// TIA Portal V15.1 export
// export: Created 2024-05-17T05:38:46.400505Z, ExportSetting WithDefaults, DisplayName Totally Integrated Automation Portal, DisplayVersion V15.1 Update 5, DisplayName TIA Portal Openness, DisplayVersion V15.1 Update 5, DisplayName SINAMICS Startdrive Advanced, DisplayVersion V15.1, DisplayName G130, G150, S120, S150, SINAMICS MV, S210, DisplayVersion V15.1, DisplayName G110M, G120, G120C, G120D, G120P, DisplayVersion V15.1, DisplayName STEP 7 Professional, DisplayVersion V15.1 Update 5, DisplayName STEP 7 Safety, DisplayVersion V15.1, DisplayName WinCC Professional, DisplayVersion V15.1 Update 5, DisplayName SIMATIC Visualization Architect, DisplayVersion V15.1
FUNCTION_BLOCK "LGBRollerDoorIO"   // FB6674, FBD
TITLE = LGBRollerDoorIO
{ S7_Optimized_Access := 'TRUE' }
VERSION : 0.1
// stored: AutoNumber false, IsIECCheckEnabled false, IsRetainMemResEnabled false, MemoryReserve 100, SetENOAutomatically False, UDAEnableTagReadback false
   VAR_INPUT
      I_DoorOpened { ExternalAccessible := 'False'; ExternalVisible := 'False'; ExternalWritable := 'False'} : Bool;   // Position Set detection or summary / Door Opened
      I_DoorClosed { ExternalAccessible := 'False'; ExternalVisible := 'False'; ExternalWritable := 'False'} : Bool;   // Position Reset detection or summary / Door Closed
      I_DoorClosedSafety { ExternalAccessible := 'False'; ExternalVisible := 'False'; ExternalWritable := 'False'} : Bool;   // Position Reset detection or summary / Door Closed Safety signal
      I_Ready { ExternalAccessible := 'False'; ExternalVisible := 'False'; ExternalWritable := 'False'} : Bool;   // Device Ready
      I_EnableAlarm { ExternalAccessible := 'False'; ExternalVisible := 'False'; ExternalWritable := 'False'} : Bool;   // Enable alarm / Enable Alarm
      I_MotorProtection { ExternalAccessible := 'False'; ExternalVisible := 'False'; ExternalWritable := 'False'} : Bool;   // Motor protection
      I_OpenBegin { ExternalAccessible := 'False'; ExternalVisible := 'False'; ExternalWritable := 'False'} : Bool;   // Function Set begin selection / Function Open begin selection
      I_CloseBegin { ExternalAccessible := 'False'; ExternalVisible := 'False'; ExternalWritable := 'False'} : Bool;   // Function Reset begin selection / Function Close begin selection
      I_CmdOpenIntlkOK { ExternalAccessible := 'False'; ExternalVisible := 'False'; ExternalWritable := 'False'} : Bool;   // Set Interlock / Command Open Interlock
      I_CmdCloseIntlkOK { ExternalAccessible := 'False'; ExternalVisible := 'False'; ExternalWritable := 'False'} : Bool;   // Reset Interlock / Command Close Interlock
      I_PBSet { ExternalAccessible := 'False'; ExternalVisible := 'False'; ExternalWritable := 'False'} : Bool;   // Push button for Set direction (used in manual with button OP panels )
      I_PBReset { ExternalAccessible := 'False'; ExternalVisible := 'False'; ExternalWritable := 'False'} : Bool;   // Push button for reset direcion (used in manual with pushbutton OP panels) / Push button for Reset direction (used in manual with Pushbutton OP panels)
      I_SafetyOk { ExternalAccessible := 'False'; ExternalVisible := 'False'; ExternalWritable := 'False'} : Bool;   // Safety Ok
      C_MotorProtectionNc { ExternalAccessible := 'False'; ExternalVisible := 'False'; ExternalWritable := 'False'} : Bool;   // Motor Protection Normally closed
      C_EnalbeRepatAlarmBypass { ExternalAccessible := 'False'; ExternalVisible := 'False'; ExternalWritable := 'False'} : Bool;   // Enable repeat alarm Bypass active
      C_RepeatAlarmBypass { ExternalAccessible := 'False'; ExternalVisible := 'False'; ExternalWritable := 'False'} : Time;   // Time to repeat alarm Bypass is active
   END_VAR
   VAR_OUTPUT
      O_CmdOpen { ExternalAccessible := 'False'; ExternalVisible := 'False'; ExternalWritable := 'False'} : Bool;   // Command to activate Set movement / Command to Activate Set movement / Command to Activate Open movement
      O_CmdClose { ExternalAccessible := 'False'; ExternalVisible := 'False'; ExternalWritable := 'False'} : Bool;   // Command to activate Reset movement / Command to Activate Reset movement / Command to Activate Close movement
      O_DoorOpened { ExternalAccessible := 'False'; ExternalVisible := 'False'; ExternalWritable := 'False'} : Bool;   // Door Opened
      O_DoorClosed { ExternalAccessible := 'False'; ExternalVisible := 'False'; ExternalWritable := 'False'} : Bool;   // Door Closed
      O_FuncRunning { ExternalAccessible := 'False'; ExternalVisible := 'False'; ExternalWritable := 'False'} : Bool;   // Signal that the function is busy
      O_LEDOpen { ExternalAccessible := 'False'; ExternalVisible := 'False'; ExternalWritable := 'False'} : Bool;   // Ledindication / Led indication for Open
      O_LEDClose { ExternalAccessible := 'False'; ExternalVisible := 'False'; ExternalWritable := 'False'} : Bool;   // Ledindication / Led indication for Close
      O_AlarmABCondition { ExternalAccessible := 'False'; ExternalVisible := 'False'; ExternalWritable := 'False'} : Bool;   // Alarms AB condition
      O_AlarmA { ExternalAccessible := 'False'; ExternalVisible := 'False'; ExternalWritable := 'False'} : Bool;   // Summation Alarm A of roller. / Alarm A
      O_AlarmB { ExternalAccessible := 'False'; ExternalVisible := 'False'; ExternalWritable := 'False'} : Bool;   // Summation Alarm B of roller. / Alarm B
      O_AlarmC { ExternalAccessible := 'False'; ExternalVisible := 'False'; ExternalWritable := 'False'} : Bool;   // Summation Alarm C of roller. / Alarm C
      O_AlarmD { ExternalAccessible := 'False'; ExternalVisible := 'False'; ExternalWritable := 'False'} : Bool;   // Summation Alarm D of roller. / Alarm D
      H_AlarmDWord { ExternalAccessible := 'False'; ExternalVisible := 'False'; ExternalWritable := 'False'} : DWord;   // HMI Animation of the alarms of the roller / HMI Animation
   END_VAR
   VAR_IN_OUT
      IO_GroupInterlock { ExternalAccessible := 'False'; ExternalVisible := 'False'; ExternalWritable := 'False'} : Bool;   // Is this OP selected? Refers to the interlocking word of this group
      IO_Modes : "Modes";
      H_HMI : "H_HMI";   // Animation
      H_RollerDoorIO : "H_GBRollerDoorIO";   // Animation
   END_VAR
   VAR
      AA_MotorProtectionAlm { ExternalAccessible := 'False'; ExternalVisible := 'False'; ExternalWritable := 'False'} : Bool;   // Motor protection alarm / Motor protection Alarm
      AB_DoorClosedSafety { ExternalAccessible := 'False'; ExternalVisible := 'False'; ExternalWritable := 'False'} : Bool;   // Safety Switch alarm / Safety Switch Alarm / Door is closed but the safety signal 'Door Closed' is missing
      AB_DoorClosedNotSafety { ExternalAccessible := 'False'; ExternalVisible := 'False'; ExternalWritable := 'False'} : Bool;   // Safety Switch alarm / Safety Switch Alarm / Door is closed but the NOT safety signal 'Door Closed' is missing
      AC_NotReadyAlm { ExternalAccessible := 'False'; ExternalVisible := 'False'; ExternalWritable := 'False'} : Bool;   // Not Ready To Run / Ej Drift Klar
      AC_OutOfUse { ExternalAccessible := 'False'; ExternalVisible := 'False'; ExternalWritable := 'False'} : Bool;   // The bypass is active, door is Out of Use (stay ALL the time open)
      AD_IntlkOpenAlm { ExternalAccessible := 'False'; ExternalVisible := 'False'; ExternalWritable := 'False'} : Bool;   // Alarm interlock Set / Alarm Interlock Set / Alarm Interlock Command Open
      AD_IntlkCloseAlm { ExternalAccessible := 'False'; ExternalVisible := 'False'; ExternalWritable := 'False'} : Bool;   // Alarm interlock Reset / Alarm Interlock Reset / Alarm Interlock Command Close
      AlarmA { ExternalAccessible := 'False'; ExternalVisible := 'False'; ExternalWritable := 'False'} : Bool;   // Summation Alarm A
      AlarmB { ExternalAccessible := 'False'; ExternalVisible := 'False'; ExternalWritable := 'False'} : Bool;   // Summation Alarm B
      AlarmC { ExternalAccessible := 'False'; ExternalVisible := 'False'; ExternalWritable := 'False'} : Bool;   // Summation Alarm C
      AlarmD { ExternalAccessible := 'False'; ExternalVisible := 'False'; ExternalWritable := 'False'} : Bool;   // Summation Alarm D
      FuncRunning { ExternalAccessible := 'False'; ExternalVisible := 'False'; ExternalWritable := 'False'} : Bool;   // Function running
      AlarmCondMotorProtection { ExternalAccessible := 'False'; ExternalVisible := 'False'; ExternalWritable := 'False'} : Bool;   // Alarm condition
      AlarmCondDoorClosedSafety { ExternalAccessible := 'False'; ExternalVisible := 'False'; ExternalWritable := 'False'} : Bool;   // Alarm condition
      AlarmCondDoorClosedNotSafety { ExternalAccessible := 'False'; ExternalVisible := 'False'; ExternalWritable := 'False'} : Bool;   // Alarm condition
      IntlkOpenAlmCond { ExternalAccessible := 'False'; ExternalVisible := 'False'; ExternalWritable := 'False'} : Bool;   // Alarm interlock Set condition / Alarm Interlock Set condition / Alarm Interlock Open condition
      IntlkCloseAlmCond { ExternalAccessible := 'False'; ExternalVisible := 'False'; ExternalWritable := 'False'} : Bool;   // Alarm interlock Reset condition / Alarm Interlock Reset condition / Alarm Interlock Close condition
      CmdOpen { ExternalAccessible := 'False'; ExternalVisible := 'False'; ExternalWritable := 'False'} : Bool;   // Command set / Command Open Door
      CmdClose { ExternalAccessible := 'False'; ExternalVisible := 'False'; ExternalWritable := 'False'} : Bool;   // Dommand reset / DCommand Reset / Command Close Door
      AlarmABCondition { ExternalAccessible := 'False'; ExternalVisible := 'False'; ExternalWritable := 'False'} : Bool;   // Alarm AB condition / Alarm AB Condition
   END_VAR
   VAR DB_SPECIFIC
      OpenCloseOutOfUse { ExternalAccessible := 'False'; ExternalVisible := 'False'; ExternalWritable := 'False'} : Bool;   // Status door by Out of Use
      Edge { ExternalAccessible := 'False'; ExternalVisible := 'False'; ExternalWritable := 'False'} : Array[0..10] of Bool;   // Edge
   END_VAR
   VAR
      T_DoorClosedSafety { ExternalAccessible := 'False'; ExternalVisible := 'False'; ExternalWritable := 'False'} : IEC_TIMER;   // On Delay Timer Safety signal
      T_DoorClosedNotSafety { ExternalAccessible := 'False'; ExternalVisible := 'False'; ExternalWritable := 'False'} : IEC_TIMER;   // On Delay Timer Safety signal
      T_RepeatAlarmOutOfUSe { ExternalAccessible := 'False'; ExternalVisible := 'False'; ExternalWritable := 'False'} : IEC_TIMER;   // On Delay Timer Repeat Alarm
   END_VAR
   VAR_TEMP
      DoorOpened : Bool;   // Set position / Set Position / Door Opened or summary
      DoorClosed : Bool;   // Reset position / Reset Position / Door Opened or summary
   END_VAR
   VAR_TEMP   // added for the SCL form of the ladder/FBD networks
      _w1 : Bool;
      _w2 : Bool;
   END_VAR
BEGIN

REGION Network 1: **** 2.2 - Alarms - Alarm Generation **** Condition for the Motor Protection Alarm
   // Condition for the Alarm Motor Protection
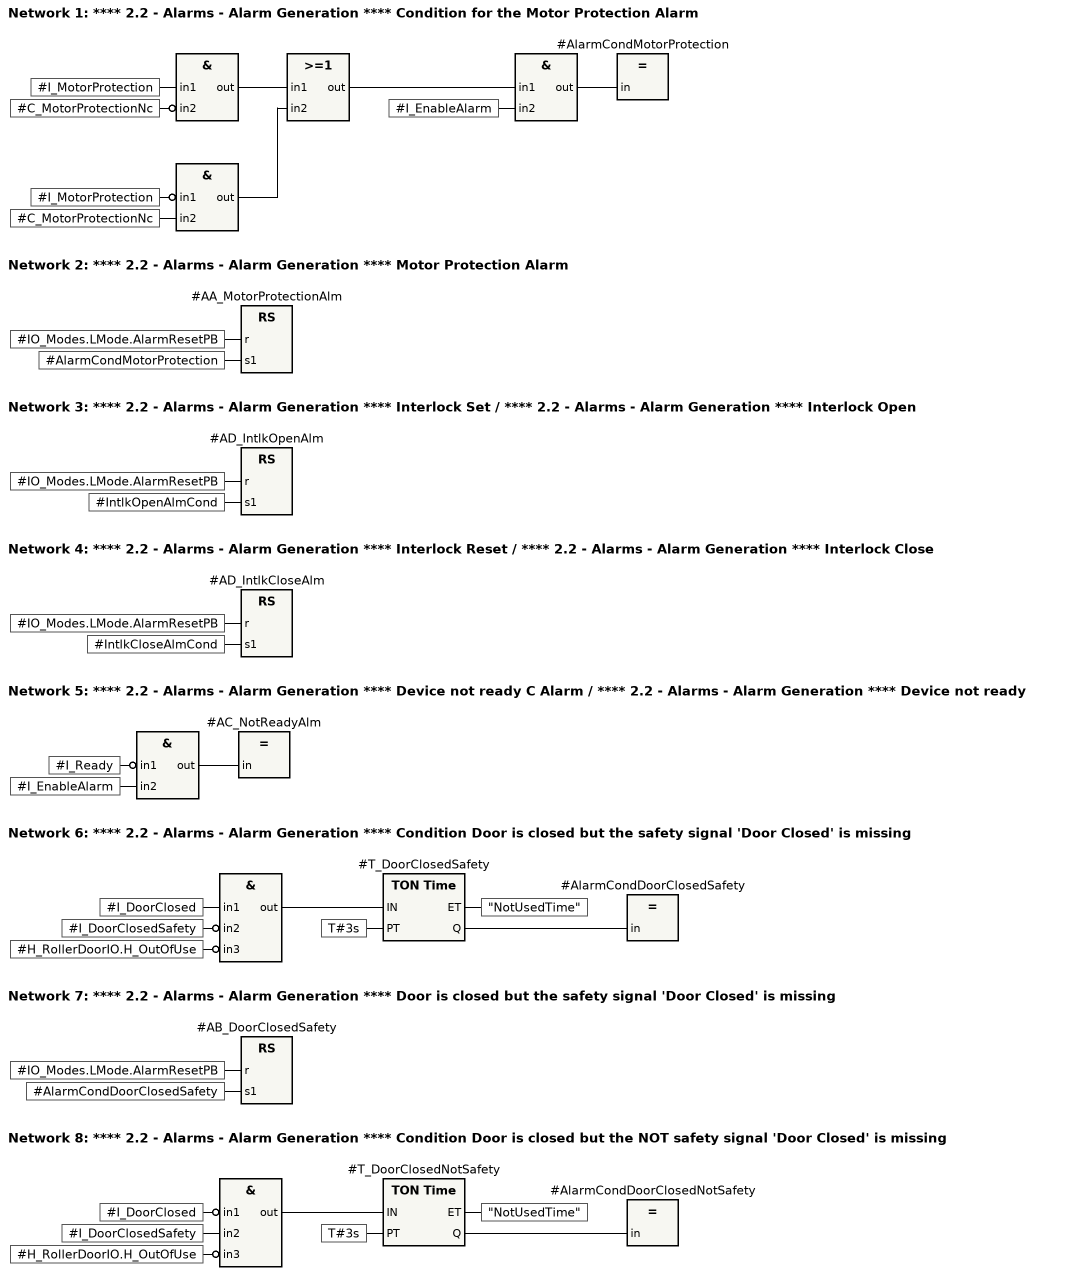
   #AlarmCondMotorProtection := ((#I_MotorProtection AND NOT #C_MotorProtectionNc) OR (NOT #I_MotorProtection AND #C_MotorProtectionNc)) AND #I_EnableAlarm;
END_REGION

REGION Network 2: **** 2.2 - Alarms - Alarm Generation **** Motor Protection Alarm
   // Motor Protection Alarm
   IF #IO_Modes.LMode.AlarmResetPB THEN
       #AA_MotorProtectionAlm := FALSE;   // RS flip-flop
   END_IF;
   IF #AlarmCondMotorProtection THEN #AA_MotorProtectionAlm := TRUE; END_IF;
END_REGION

REGION Network 3: **** 2.2 - Alarms - Alarm Generation **** Interlock Set / **** 2.2 - Alarms - Alarm Generation **** Interlock Open
   // Interlock Set / Interlock Open
   IF #IO_Modes.LMode.AlarmResetPB THEN
       #AD_IntlkOpenAlm := FALSE;   // RS flip-flop
   END_IF;
   IF #IntlkOpenAlmCond THEN #AD_IntlkOpenAlm := TRUE; END_IF;
END_REGION

REGION Network 4: **** 2.2 - Alarms - Alarm Generation **** Interlock Reset / **** 2.2 - Alarms - Alarm Generation **** Interlock Close
   // Interlock Reset / Interlock Close
   IF #IO_Modes.LMode.AlarmResetPB THEN
       #AD_IntlkCloseAlm := FALSE;   // RS flip-flop
   END_IF;
   IF #IntlkCloseAlmCond THEN #AD_IntlkCloseAlm := TRUE; END_IF;
END_REGION

REGION Network 5: **** 2.2 - Alarms - Alarm Generation **** Device not ready C Alarm / **** 2.2 - Alarms - Alarm Generation **** Device not ready
   // Device not ready C Alarm
   #AC_NotReadyAlm := NOT #I_Ready AND #I_EnableAlarm;
END_REGION

REGION Network 6: **** 2.2 - Alarms - Alarm Generation **** Condition Door is closed but the safety signal 'Door Closed' is missing
   #T_DoorClosedSafety.TON(IN := #I_DoorClosed AND NOT #I_DoorClosedSafety AND NOT #H_RollerDoorIO.H_OutOfUse,
                           PT := T#3s,
                           ET => "NotUsedTime");
   #AlarmCondDoorClosedSafety := #T_DoorClosedSafety.Q;
END_REGION

REGION Network 7: **** 2.2 - Alarms - Alarm Generation **** Door is closed but the safety signal 'Door Closed' is missing
   IF #IO_Modes.LMode.AlarmResetPB THEN
       #AB_DoorClosedSafety := FALSE;   // RS flip-flop
   END_IF;
   IF #AlarmCondDoorClosedSafety THEN #AB_DoorClosedSafety := TRUE; END_IF;
END_REGION

REGION Network 8: **** 2.2 - Alarms - Alarm Generation **** Condition Door is closed but the NOT safety signal 'Door Closed' is missing
   #T_DoorClosedNotSafety.TON(IN := NOT #I_DoorClosed AND #I_DoorClosedSafety AND NOT #H_RollerDoorIO.H_OutOfUse,
                           PT := T#3s,
                           ET => "NotUsedTime");
   #AlarmCondDoorClosedNotSafety := #T_DoorClosedNotSafety.Q;
END_REGION

REGION Network 9: **** 2.2 - Alarms - Alarm Generation **** Door is closed but the safety signal 'Door Closed' is missing
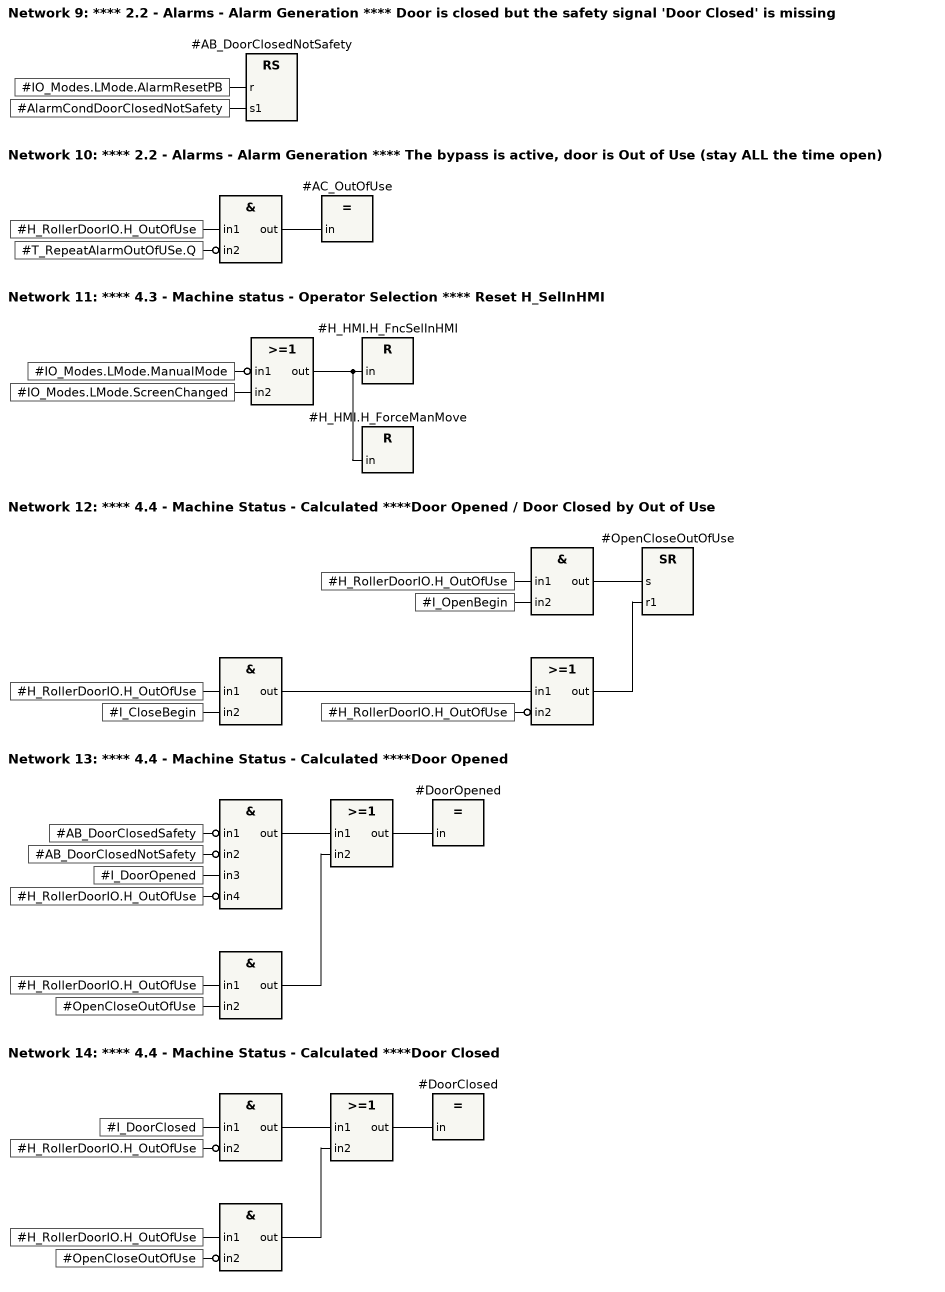
   IF #IO_Modes.LMode.AlarmResetPB THEN
       #AB_DoorClosedNotSafety := FALSE;   // RS flip-flop
   END_IF;
   IF #AlarmCondDoorClosedNotSafety THEN #AB_DoorClosedNotSafety := TRUE; END_IF;
END_REGION

REGION Network 10: **** 2.2 - Alarms - Alarm Generation **** The bypass is active, door is Out of Use (stay ALL the time open)
   #AC_OutOfUse := #H_RollerDoorIO.H_OutOfUse AND NOT #T_RepeatAlarmOutOfUSe.Q;
END_REGION

REGION Network 11: **** 4.3 - Machine status - Operator Selection **** Reset H_SelInHMI
   // Reset H_SelInHMI
   IF NOT #IO_Modes.LMode.ManualMode OR #IO_Modes.LMode.ScreenChanged THEN
       #H_HMI.H_FncSelInHMI := FALSE;
       #H_HMI.H_ForceManMove := FALSE;
   END_IF;
END_REGION

REGION Network 12: **** 4.4 - Machine Status - Calculated ****Door Opened / Door Closed by Out of Use
   IF #H_RollerDoorIO.H_OutOfUse AND #I_OpenBegin THEN
       #OpenCloseOutOfUse := TRUE;   // SR flip-flop
   END_IF;
   IF (#H_RollerDoorIO.H_OutOfUse AND #I_CloseBegin) OR NOT #H_RollerDoorIO.H_OutOfUse THEN
       #OpenCloseOutOfUse := FALSE;
   END_IF;
END_REGION

REGION Network 13: **** 4.4 - Machine Status - Calculated ****Door Opened
   // Albany Roller Door Opened
   #DoorOpened := (NOT #AB_DoorClosedSafety AND NOT #AB_DoorClosedNotSafety AND #I_DoorOpened AND NOT #H_RollerDoorIO.H_OutOfUse) OR (#H_RollerDoorIO.H_OutOfUse AND #OpenCloseOutOfUse);
END_REGION

REGION Network 14: **** 4.4 - Machine Status - Calculated ****Door Closed
   // Albany Roller Door Closed
   #DoorClosed := (#I_DoorClosed AND NOT #H_RollerDoorIO.H_OutOfUse) OR (#H_RollerDoorIO.H_OutOfUse AND NOT #OpenCloseOutOfUse);
END_REGION

REGION Network 15: **** 4.6 - Machine Status - Indication **** Motor Loop Animation / **** 4.6 - Machine Status - Indication **** Icon Animation
   // Motor Loop Animation / Icon Animation
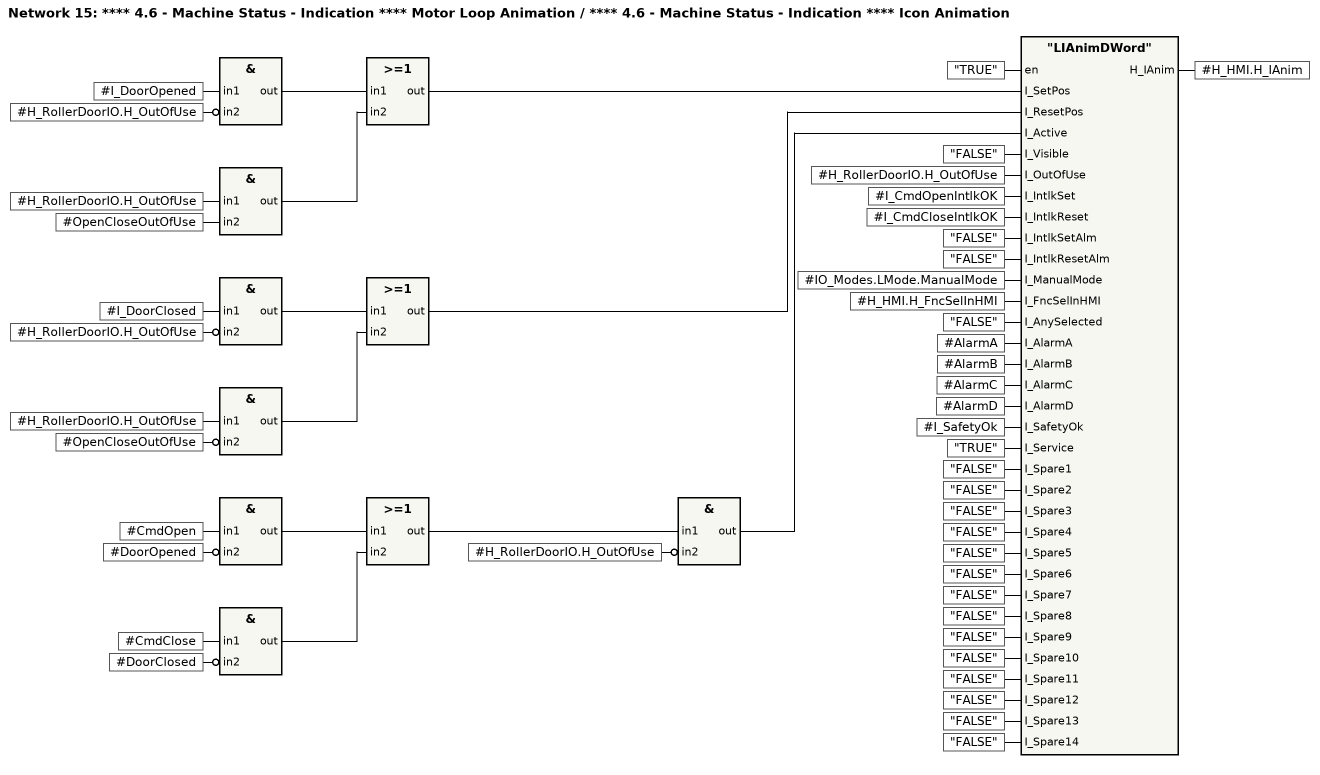
   IF "TRUE" THEN
       "LIAnimDWord"(I_SetPos := (#I_DoorOpened AND NOT #H_RollerDoorIO.H_OutOfUse) OR (#H_RollerDoorIO.H_OutOfUse AND #OpenCloseOutOfUse),
                     I_ResetPos := (#I_DoorClosed AND NOT #H_RollerDoorIO.H_OutOfUse) OR (#H_RollerDoorIO.H_OutOfUse AND NOT #OpenCloseOutOfUse),
                     I_Active := ((#CmdOpen AND NOT #DoorOpened) OR (#CmdClose AND NOT #DoorClosed)) AND NOT #H_RollerDoorIO.H_OutOfUse,
                     I_Visible := "FALSE",
                     I_OutOfUse := #H_RollerDoorIO.H_OutOfUse,
                     I_IntlkSet := #I_CmdOpenIntlkOK,
                     I_IntlkReset := #I_CmdCloseIntlkOK,
                     I_IntlkSetAlm := "FALSE",
                     I_IntlkResetAlm := "FALSE",
                     I_ManualMode := #IO_Modes.LMode.ManualMode,
                     I_FncSelInHMI := #H_HMI.H_FncSelInHMI,
                     I_AnySelected := "FALSE",
                     I_AlarmA := #AlarmA,
                     I_AlarmB := #AlarmB,
                     I_AlarmC := #AlarmC,
                     I_AlarmD := #AlarmD,
                     I_SafetyOk := #I_SafetyOk,
                     I_Service := "TRUE",
                     I_Spare1 := "FALSE",
                     I_Spare2 := "FALSE",
                     I_Spare3 := "FALSE",
                     I_Spare4 := "FALSE",
                     I_Spare5 := "FALSE",
                     I_Spare6 := "FALSE",
                     I_Spare7 := "FALSE",
                     I_Spare8 := "FALSE",
                     I_Spare9 := "FALSE",
                     I_Spare10 := "FALSE",
                     I_Spare11 := "FALSE",
                     I_Spare12 := "FALSE",
                     I_Spare13 := "FALSE",
                     I_Spare14 := "FALSE",
                     H_IAnim => #H_HMI.H_IAnim);
   END_IF;
END_REGION

REGION Network 16: **** 4.6 - Machine Status - Indication **** Animation
   // Animation
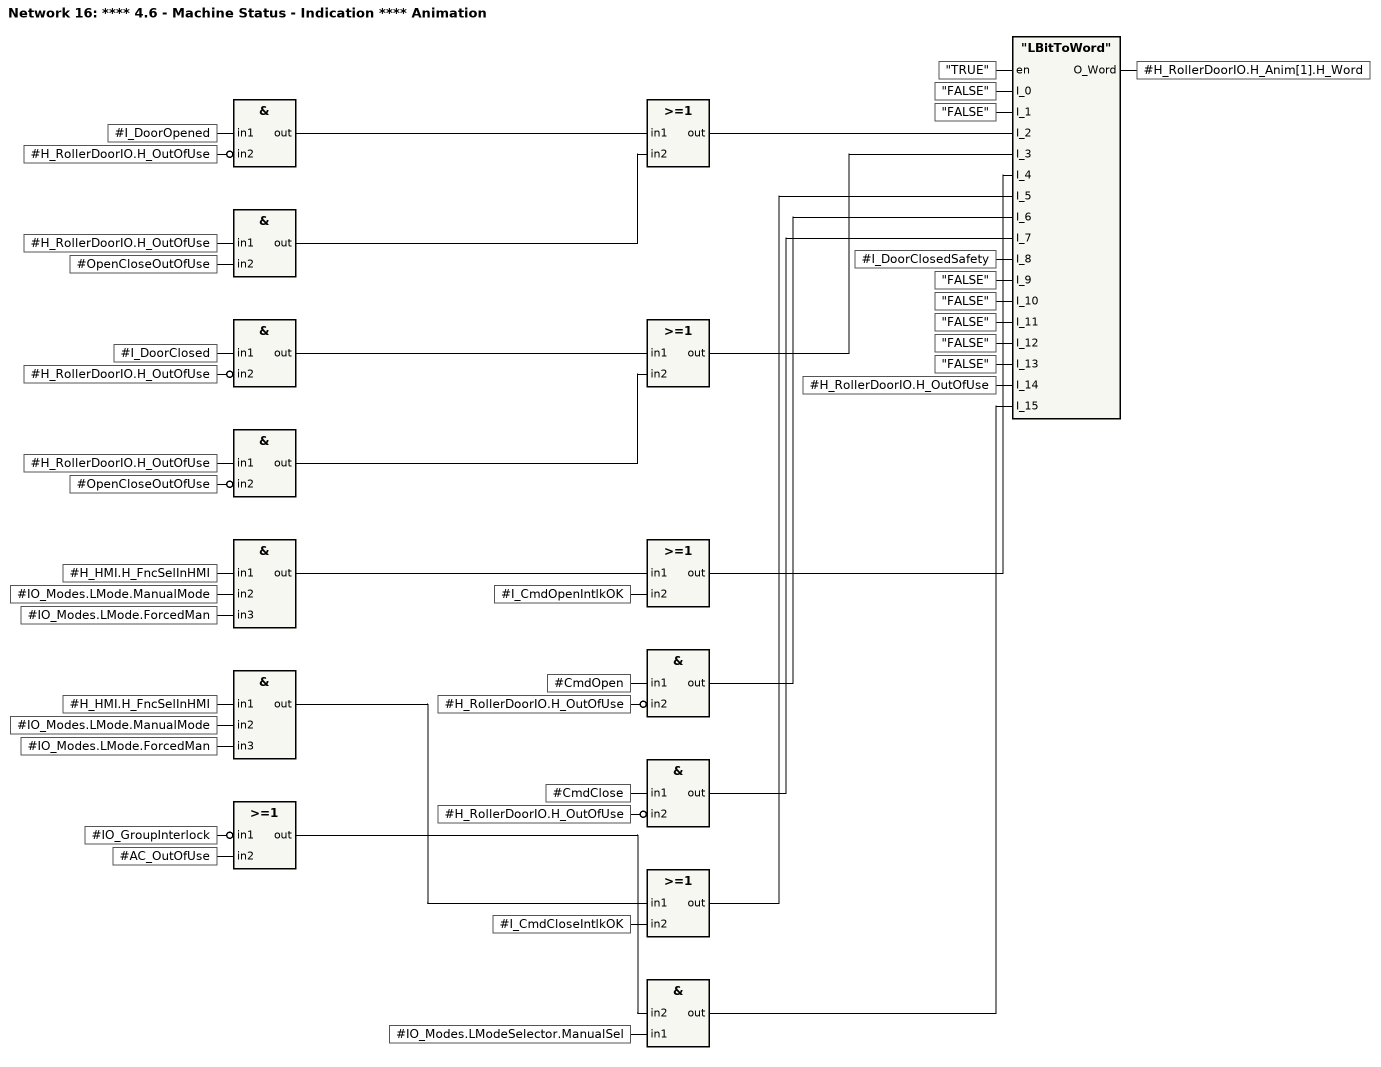
   IF "TRUE" THEN
       "LBitToWord"(I_0 := "FALSE",
                    I_1 := "FALSE",
                    I_2 := (#I_DoorOpened AND NOT #H_RollerDoorIO.H_OutOfUse) OR (#H_RollerDoorIO.H_OutOfUse AND #OpenCloseOutOfUse),
                    I_3 := (#I_DoorClosed AND NOT #H_RollerDoorIO.H_OutOfUse) OR (#H_RollerDoorIO.H_OutOfUse AND NOT #OpenCloseOutOfUse),
                    I_4 := (#H_HMI.H_FncSelInHMI AND #IO_Modes.LMode.ManualMode AND #IO_Modes.LMode.ForcedMan) OR #I_CmdOpenIntlkOK,
                    I_5 := (#H_HMI.H_FncSelInHMI AND #IO_Modes.LMode.ManualMode AND #IO_Modes.LMode.ForcedMan) OR #I_CmdCloseIntlkOK,
                    I_6 := #CmdOpen AND NOT #H_RollerDoorIO.H_OutOfUse,
                    I_7 := #CmdClose AND NOT #H_RollerDoorIO.H_OutOfUse,
                    I_8 := #I_DoorClosedSafety,
                    I_9 := "FALSE",
                    I_10 := "FALSE",
                    I_11 := "FALSE",
                    I_12 := "FALSE",
                    I_13 := "FALSE",
                    I_14 := #H_RollerDoorIO.H_OutOfUse,
                    I_15 := (NOT #IO_GroupInterlock OR #AC_OutOfUse) AND #IO_Modes.LModeSelector.ManualSel,
                    O_Word => #H_RollerDoorIO.H_Anim[1].H_Word);
   END_IF;
END_REGION

REGION Network 17: **** 4.6 - Machine Status - Indication **** Animation
   // Animation
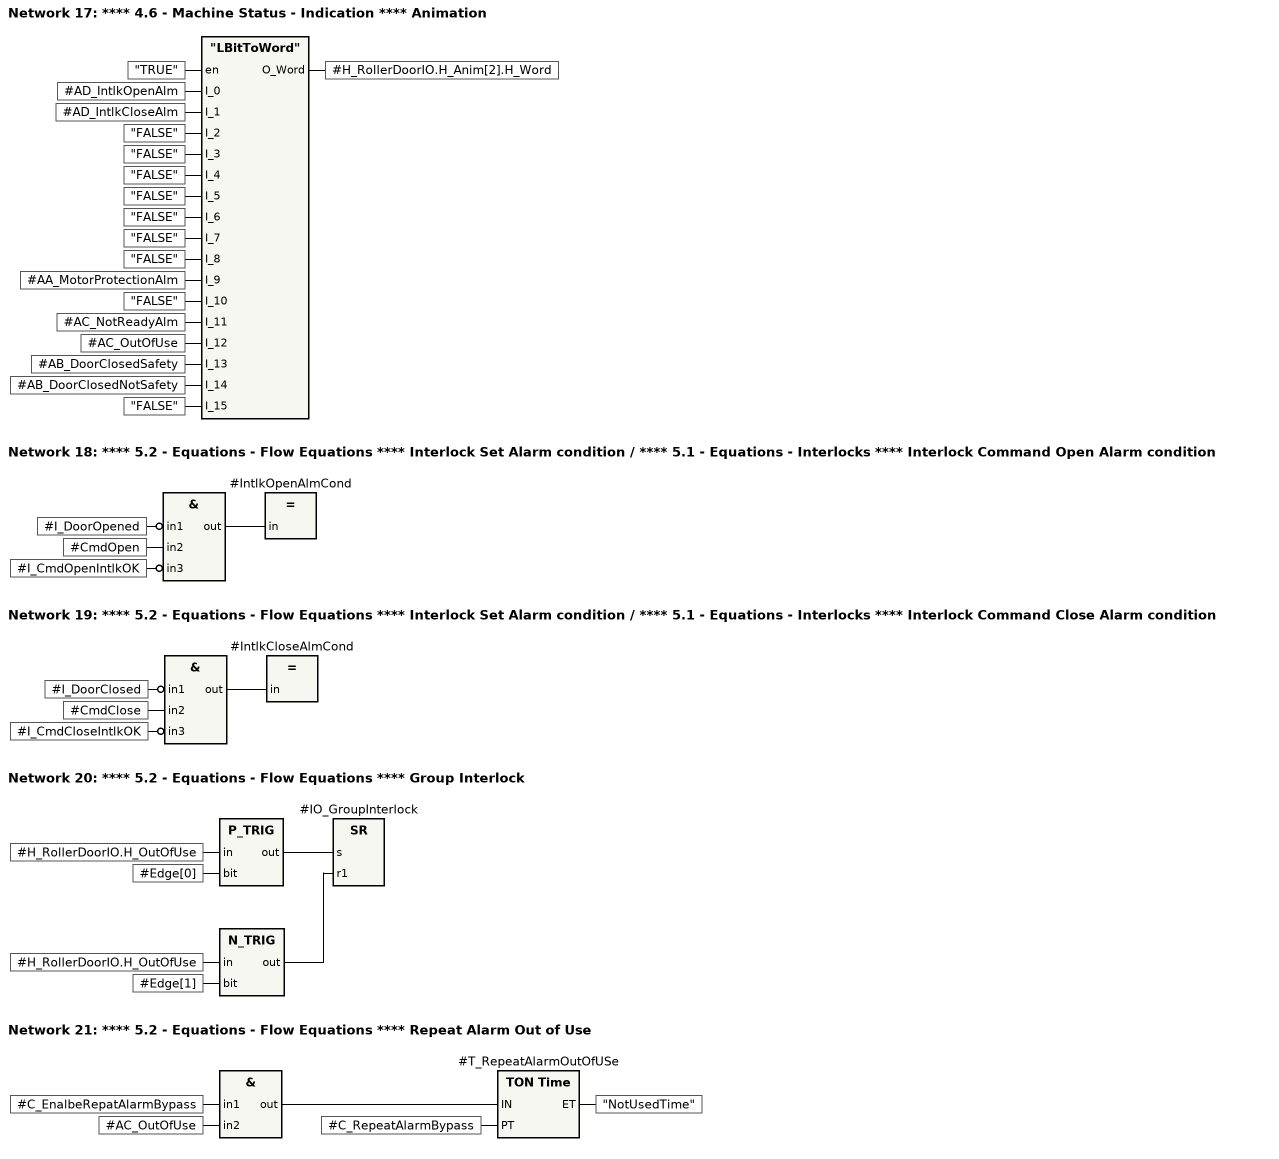
   IF "TRUE" THEN
       "LBitToWord"(I_0 := #AD_IntlkOpenAlm,
                    I_1 := #AD_IntlkCloseAlm,
                    I_2 := "FALSE",
                    I_3 := "FALSE",
                    I_4 := "FALSE",
                    I_5 := "FALSE",
                    I_6 := "FALSE",
                    I_7 := "FALSE",
                    I_8 := "FALSE",
                    I_9 := #AA_MotorProtectionAlm,
                    I_10 := "FALSE",
                    I_11 := #AC_NotReadyAlm,
                    I_12 := #AC_OutOfUse,
                    I_13 := #AB_DoorClosedSafety,
                    I_14 := #AB_DoorClosedNotSafety,
                    I_15 := "FALSE",
                    O_Word => #H_RollerDoorIO.H_Anim[2].H_Word);
   END_IF;
END_REGION

REGION Network 18: **** 5.2 - Equations - Flow Equations **** Interlock Set Alarm condition / **** 5.1 - Equations - Interlocks **** Interlock Command Open Alarm condition
   // Interlock Set Alarm condition / Interlock Command Open Alarm condition
   #IntlkOpenAlmCond := NOT #I_DoorOpened AND #CmdOpen AND NOT #I_CmdOpenIntlkOK;
END_REGION

REGION Network 19: **** 5.2 - Equations - Flow Equations **** Interlock Set Alarm condition / **** 5.1 - Equations - Interlocks **** Interlock Command Close Alarm condition
   // Interlock Set Alarm condition / Interlock Command Close Alarm condition
   #IntlkCloseAlmCond := NOT #I_DoorClosed AND #CmdClose AND NOT #I_CmdCloseIntlkOK;
END_REGION

REGION Network 20: **** 5.2 - Equations - Flow Equations **** Group Interlock
   #_w1 := #H_RollerDoorIO.H_OutOfUse AND NOT #Edge[0];   // rising edge
   #Edge[0] := #H_RollerDoorIO.H_OutOfUse;
   #_w2 := NOT #H_RollerDoorIO.H_OutOfUse AND #Edge[1];   // falling edge
   #Edge[1] := #H_RollerDoorIO.H_OutOfUse;
   IF #_w1 THEN
       #IO_GroupInterlock := TRUE;   // SR flip-flop
   END_IF;
   IF #_w2 THEN #IO_GroupInterlock := FALSE; END_IF;
END_REGION

REGION Network 21: **** 5.2 - Equations - Flow Equations **** Repeat Alarm Out of Use
   #T_RepeatAlarmOutOfUSe.TON(IN := #C_EnalbeRepatAlarmBypass AND #AC_OutOfUse,
                           PT := #C_RepeatAlarmBypass,
                           ET => "NotUsedTime");
END_REGION

REGION Network 22: **** 5.2 - Equations - Flow Equations **** Open Door
   // Open Door
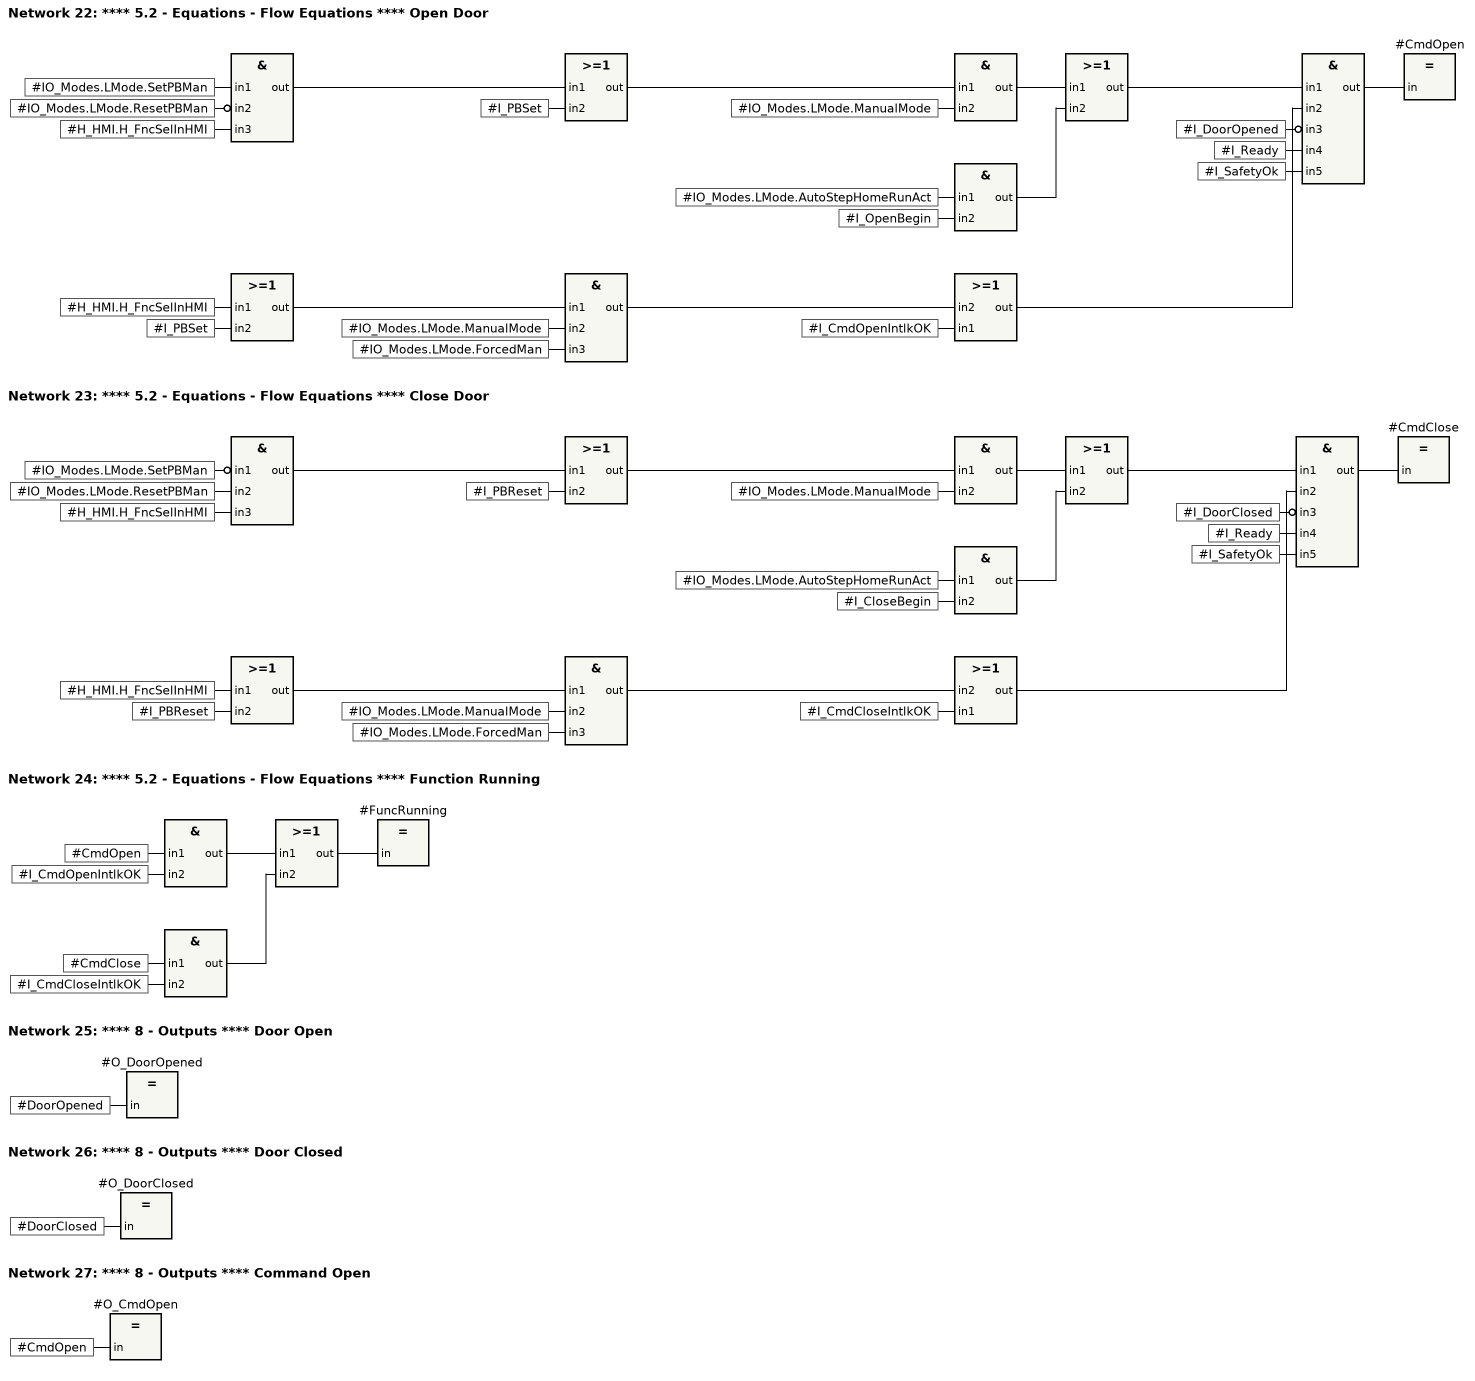
   #CmdOpen := ((((#IO_Modes.LMode.SetPBMan AND NOT #IO_Modes.LMode.ResetPBMan AND #H_HMI.H_FncSelInHMI) OR #I_PBSet) AND #IO_Modes.LMode.ManualMode) OR (#IO_Modes.LMode.AutoStepHomeRunAct AND #I_OpenBegin)) AND (((#H_HMI.H_FncSelInHMI OR #I_PBSet) AND #IO_Modes.LMode.ManualMode AND #IO_Modes.LMode.ForcedMan) OR #I_CmdOpenIntlkOK) AND NOT #I_DoorOpened AND #I_Ready AND #I_SafetyOk;
END_REGION

REGION Network 23: **** 5.2 - Equations - Flow Equations **** Close Door
   // Close Door
   #CmdClose := ((((NOT #IO_Modes.LMode.SetPBMan AND #IO_Modes.LMode.ResetPBMan AND #H_HMI.H_FncSelInHMI) OR #I_PBReset) AND #IO_Modes.LMode.ManualMode) OR (#IO_Modes.LMode.AutoStepHomeRunAct AND #I_CloseBegin)) AND (((#H_HMI.H_FncSelInHMI OR #I_PBReset) AND #IO_Modes.LMode.ManualMode AND #IO_Modes.LMode.ForcedMan) OR #I_CmdCloseIntlkOK) AND NOT #I_DoorClosed AND #I_Ready AND #I_SafetyOk;
END_REGION

REGION Network 24: **** 5.2 - Equations - Flow Equations **** Function Running
   // Function Running
   #FuncRunning := (#CmdOpen AND #I_CmdOpenIntlkOK) OR (#CmdClose AND #I_CmdCloseIntlkOK);
END_REGION

REGION Network 25: **** 8 - Outputs **** Door Open
   // Door Open
   #O_DoorOpened := #DoorOpened;
END_REGION

REGION Network 26: **** 8 - Outputs **** Door Closed
   // Door Closed
   #O_DoorClosed := #DoorClosed;
END_REGION

REGION Network 27: **** 8 - Outputs **** Command Open
   // Command Open
   #O_CmdOpen := #CmdOpen;
END_REGION

REGION Network 28: **** 8 - Outputs **** Command Close
   // Command Close
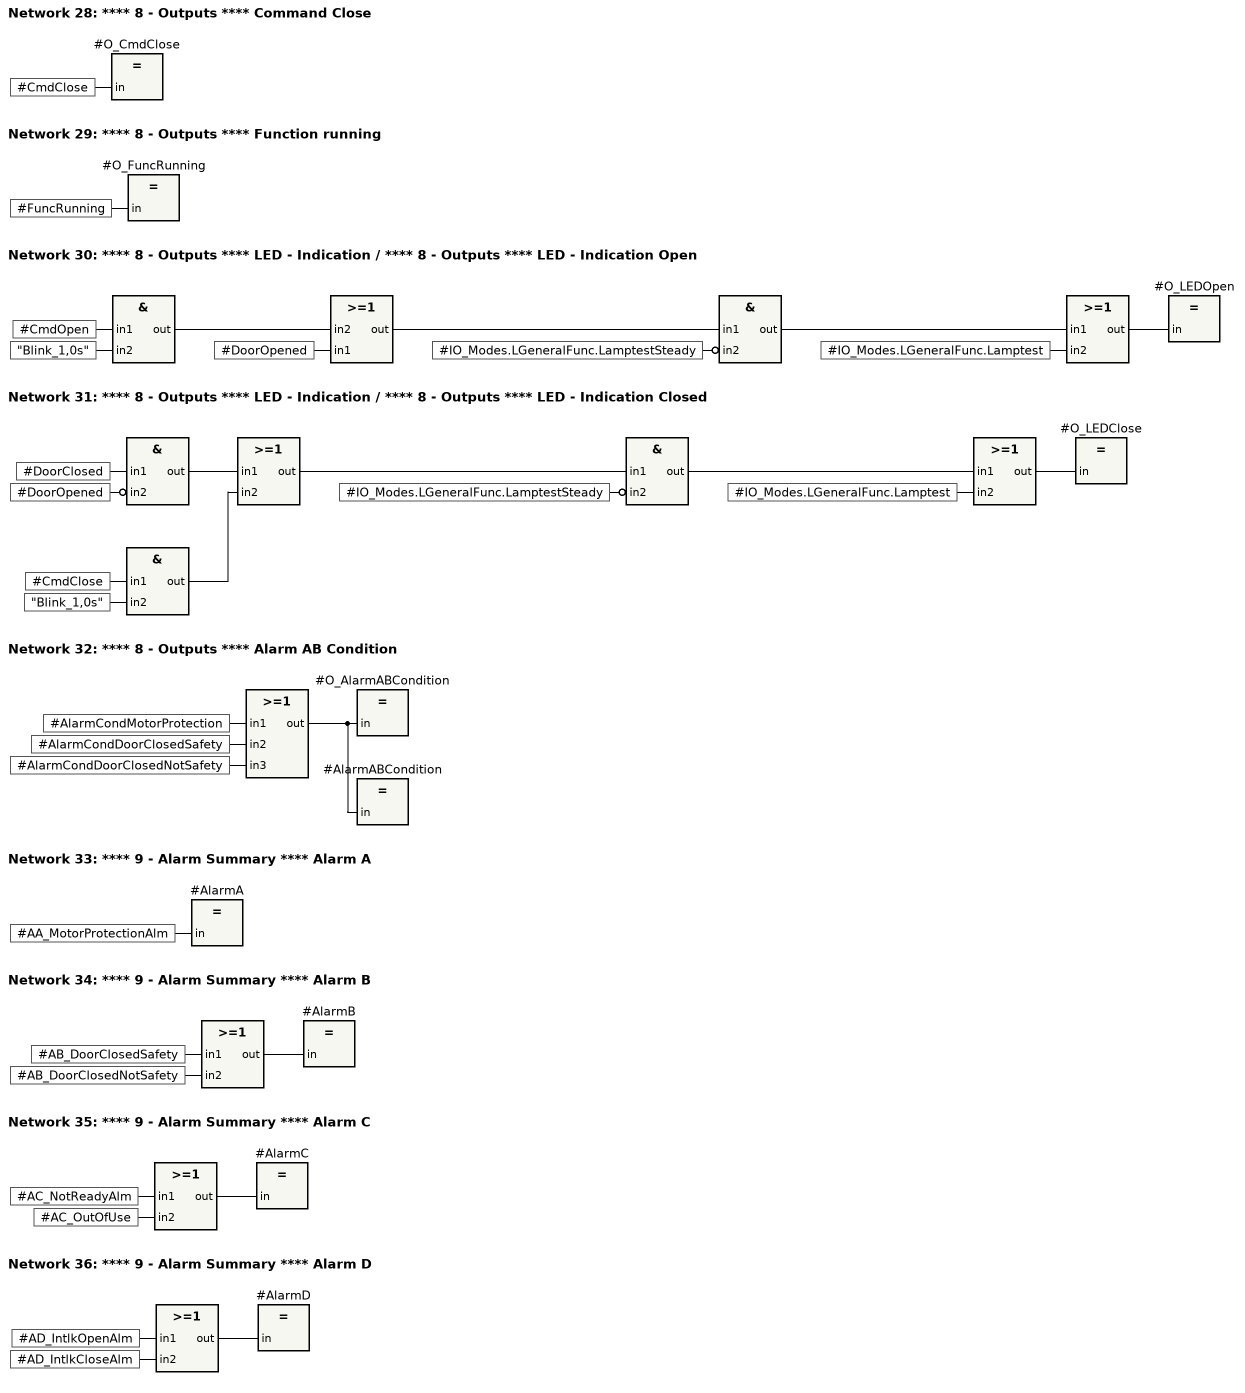
   #O_CmdClose := #CmdClose;
END_REGION

REGION Network 29: **** 8 - Outputs **** Function running
   // Function running
   #O_FuncRunning := #FuncRunning;
END_REGION

REGION Network 30: **** 8 - Outputs **** LED - Indication / **** 8 - Outputs **** LED - Indication Open
   // LED - Indication
   #O_LEDOpen := (((#CmdOpen AND "Blink_1,0s") OR #DoorOpened) AND NOT #IO_Modes.LGeneralFunc.LamptestSteady) OR #IO_Modes.LGeneralFunc.Lamptest;
END_REGION

REGION Network 31: **** 8 - Outputs **** LED - Indication / **** 8 - Outputs **** LED - Indication Closed
   // LED - Indication
   #O_LEDClose := (((#DoorClosed AND NOT #DoorOpened) OR (#CmdClose AND "Blink_1,0s")) AND NOT #IO_Modes.LGeneralFunc.LamptestSteady) OR #IO_Modes.LGeneralFunc.Lamptest;
END_REGION

REGION Network 32: **** 8 - Outputs **** Alarm AB Condition
   // Alarm AB Condition
   #O_AlarmABCondition := #AlarmCondMotorProtection OR #AlarmCondDoorClosedSafety OR #AlarmCondDoorClosedNotSafety;
   #AlarmABCondition := #O_AlarmABCondition;
END_REGION

REGION Network 33: **** 9 - Alarm Summary **** Alarm A
   // Alarms A
   #AlarmA := #AA_MotorProtectionAlm;
END_REGION

REGION Network 34: **** 9 - Alarm Summary **** Alarm B
   // Alarms B
   #AlarmB := #AB_DoorClosedSafety OR #AB_DoorClosedNotSafety;
END_REGION

REGION Network 35: **** 9 - Alarm Summary **** Alarm C
   // Alarms C
   #AlarmC := #AC_NotReadyAlm OR #AC_OutOfUse;
END_REGION

REGION Network 36: **** 9 - Alarm Summary **** Alarm D
   // Alarms D
   #AlarmD := #AD_IntlkOpenAlm OR #AD_IntlkCloseAlm;
END_REGION

REGION Network 37: **** 9 - Alarm Summary **** Alarms To Alarm UDT Alarms To Alarm UDT Get Name
   // Alarm / Alarm D
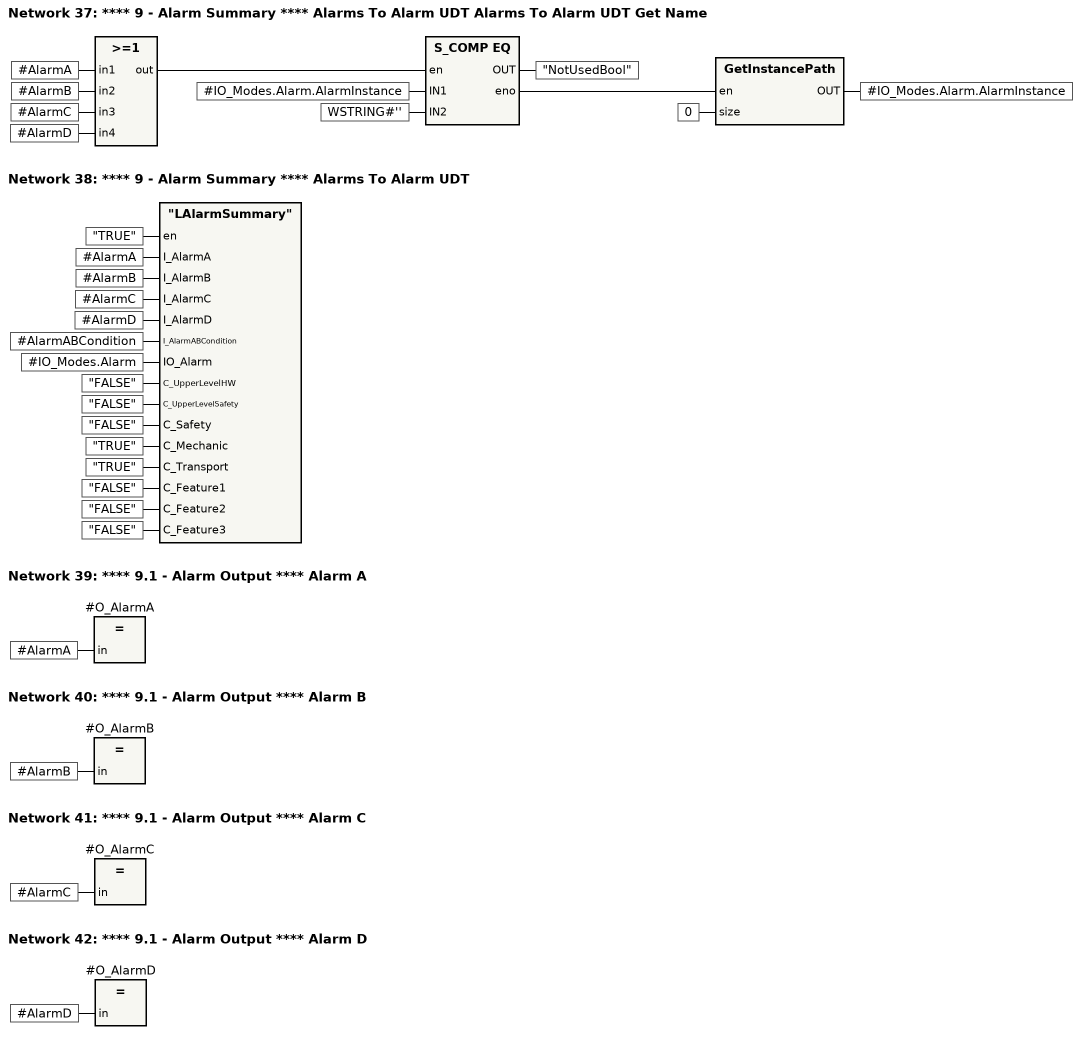
   S_COMP(EN := #AlarmA OR #AlarmB OR #AlarmC OR #AlarmD,
          IN1 := #IO_Modes.Alarm.AlarmInstance,
          IN2 := WSTRING#'',
          OUT => "NotUsedBool",
          ENO => #_w1);
   IF #_w1 THEN GetInstancePath(size := 0, OUT => #IO_Modes.Alarm.AlarmInstance); END_IF;
END_REGION

REGION Network 38: **** 9 - Alarm Summary **** Alarms To Alarm UDT
   // Alarm / Alarm D
   IF "TRUE" THEN
       "LAlarmSummary"(I_AlarmA := #AlarmA,
                       I_AlarmB := #AlarmB,
                       I_AlarmC := #AlarmC,
                       I_AlarmD := #AlarmD,
                       I_AlarmABCondition := #AlarmABCondition,
                       IO_Alarm := #IO_Modes.Alarm,
                       C_UpperLevelHW := "FALSE",
                       C_UpperLevelSafety := "FALSE",
                       C_Safety := "FALSE",
                       C_Mechanic := "TRUE",
                       C_Transport := "TRUE",
                       C_Feature1 := "FALSE",
                       C_Feature2 := "FALSE",
                       C_Feature3 := "FALSE");
   END_IF;
END_REGION

REGION Network 39: **** 9.1 - Alarm Output **** Alarm A
   // Alarms A
   #O_AlarmA := #AlarmA;
END_REGION

REGION Network 40: **** 9.1 - Alarm Output **** Alarm B
   // Alarms B
   #O_AlarmB := #AlarmB;
END_REGION

REGION Network 41: **** 9.1 - Alarm Output **** Alarm C
   // Alarms C
   #O_AlarmC := #AlarmC;
END_REGION

REGION Network 42: **** 9.1 - Alarm Output **** Alarm D
   // Alarms D
   #O_AlarmD := #AlarmD;
END_REGION

REGION Network 43: **** 9.2 - Alarm DWord**** Alarm To DWord
   // Alarm To DWord
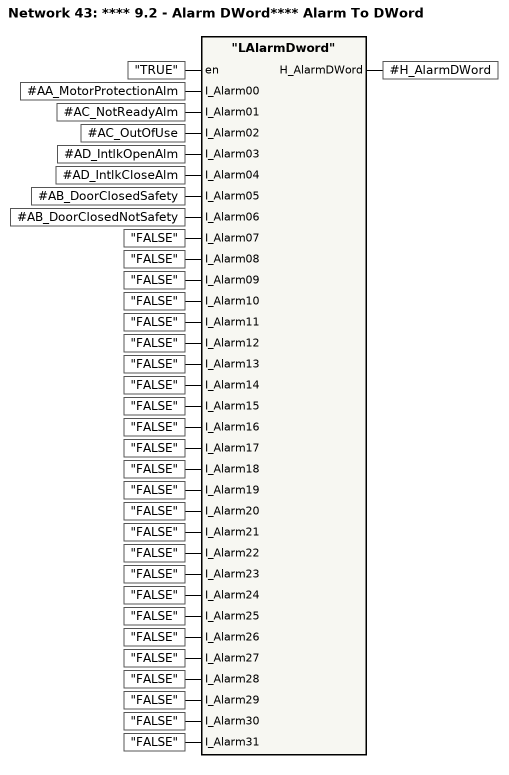
   IF "TRUE" THEN
       "LAlarmDword"(I_Alarm00 := #AA_MotorProtectionAlm,
                     I_Alarm01 := #AC_NotReadyAlm,
                     I_Alarm02 := #AC_OutOfUse,
                     I_Alarm03 := #AD_IntlkOpenAlm,
                     I_Alarm04 := #AD_IntlkCloseAlm,
                     I_Alarm05 := #AB_DoorClosedSafety,
                     I_Alarm06 := #AB_DoorClosedNotSafety,
                     I_Alarm07 := "FALSE",
                     I_Alarm08 := "FALSE",
                     I_Alarm09 := "FALSE",
                     I_Alarm10 := "FALSE",
                     I_Alarm11 := "FALSE",
                     I_Alarm12 := "FALSE",
                     I_Alarm13 := "FALSE",
                     I_Alarm14 := "FALSE",
                     I_Alarm15 := "FALSE",
                     I_Alarm16 := "FALSE",
                     I_Alarm17 := "FALSE",
                     I_Alarm18 := "FALSE",
                     I_Alarm19 := "FALSE",
                     I_Alarm20 := "FALSE",
                     I_Alarm21 := "FALSE",
                     I_Alarm22 := "FALSE",
                     I_Alarm23 := "FALSE",
                     I_Alarm24 := "FALSE",
                     I_Alarm25 := "FALSE",
                     I_Alarm26 := "FALSE",
                     I_Alarm27 := "FALSE",
                     I_Alarm28 := "FALSE",
                     I_Alarm29 := "FALSE",
                     I_Alarm30 := "FALSE",
                     I_Alarm31 := "FALSE",
                     H_AlarmDWord => #H_AlarmDWord);
   END_IF;
END_REGION
END_FUNCTION_BLOCK
